FUNCTION_BLOCK Desinfeccao (* Composite Function Block Type *)
  (* Standard: 61499-2 *)
  (* Version 0.0, 02/03/2026, template *)
  PACKAGE Hidryco.HidrycoLib;
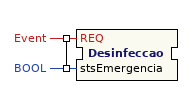
  EVENT_INPUT
    REQ WITH stsEmergencia;
  END_EVENT
  VAR_INPUT
    stsEmergencia : BOOL;
  END_VAR
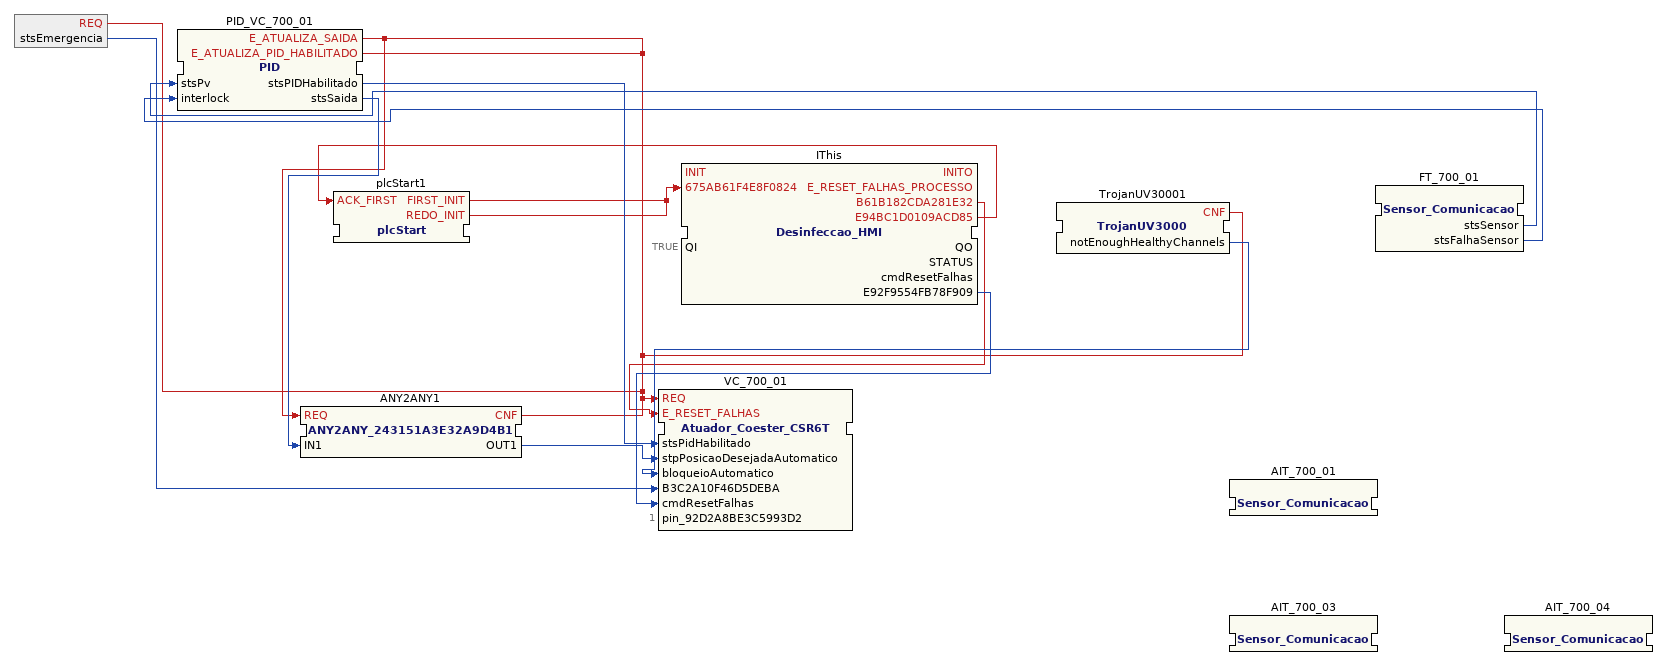
  FBS
    TrojanUV30001 : TrojanUV3000;
    VC_700_01 : Atuador_Coester_CSR6T(pin_92D2A8BE3C5993D2 := 1);
    FT_700_01 : Sensor_Comunicacao;
    AIT_700_01 : Sensor_Comunicacao;
    PID_VC_700_01 : PID;
    ANY2ANY1 : ANY2ANY_243151A3E32A9D4B1; {SET_ATTRIBUTE(Configuration.GenericFBType.InterfaceParams, Runtime.Standard#CNT:=1;IN${CNT$}:REAL;OUT${CNT$}:INT)}
    AIT_700_04 : Sensor_Comunicacao;
    AIT_700_03 : Sensor_Comunicacao;
    IThis : Desinfeccao_HMI(QI := TRUE);
    plcStart1 : plcStart;
  END_FBS
  EVENT_CONNECTIONS
    PID_VC_700_01.E_ATUALIZA_SAIDA TO VC_700_01.REQ;
    PID_VC_700_01.E_ATUALIZA_PID_HABILITADO TO VC_700_01.REQ;
    PID_VC_700_01.E_ATUALIZA_SAIDA TO ANY2ANY1.REQ;
    ANY2ANY1.CNF TO VC_700_01.REQ;
    TrojanUV30001.CNF TO VC_700_01.REQ;
    REQ TO VC_700_01.REQ;
    plcStart1.FIRST_INIT TO IThis.675AB61F4E8F0824;
    plcStart1.REDO_INIT TO IThis.675AB61F4E8F0824;
    IThis.B61B182CDA281E32 TO VC_700_01.E_RESET_FALHAS;
    IThis.E94BC1D0109ACD85 TO plcStart1.ACK_FIRST;
  END_CONNECTIONS
  DATA_CONNECTIONS
    PID_VC_700_01.stsPIDHabilitado TO VC_700_01.stsPidHabilitado;
    PID_VC_700_01.stsSaida TO ANY2ANY1.IN1;
    ANY2ANY1.OUT1 TO VC_700_01.stpPosicaoDesejadaAutomatico;
    FT_700_01.stsSensor TO PID_VC_700_01.stsPv;
    FT_700_01.stsFalhaSensor TO PID_VC_700_01.interlock;
    TrojanUV30001.notEnoughHealthyChannels TO VC_700_01.bloqueioAutomatico;
    stsEmergencia TO VC_700_01.B3C2A10F46D5DEBA;
    IThis.E92F9554FB78F909 TO VC_700_01.cmdResetFalhas;
  END_CONNECTIONS
END_FUNCTION_BLOCK
